// TIA Portal V20 export
FUNCTION_BLOCK "FB_FixtureUnloadLoad"   // FB65, SCL
{ S7_Optimized_Access := 'TRUE' }
// stored: MemoryReserve 100, SetENOAutomatically false
   VAR_INPUT
      iFixtureUnloadingRequest : Bool;
      iFixtureLoadingRequest : Bool;
      iFixtureBlowingRequest : Bool;
      iFixtureReleaseRequest : Bool;
      iFixtureV_InitRequest : Bool;
      iFixtureW_InitRequest : Bool;
      iWorkingModeFilling : Bool;
      iWorkingModeEmptying : Bool;
      iGripperReadyForUnloading : Bool;
      iGripperReadyForLoading : Bool;
      iGripperReadyForBlowing : Bool;
      iGripperReadyForRelease : Bool;
      iGripperReadyForV_Init : Bool;
      iGripperReadyForW_Init : Bool;
      iFixtureReadyForUnloading : Bool;
      iFixtureReadyForLoading : Bool;
      iFixtureReadyForBlowing : Bool;
      iFixtureReadyForRelease : Bool;
      iFixtureReadyForV_Init : Bool;
      iFixtureReadyForW_Init : Bool;
      iAxisReadyForUnloading : Bool;
      iAxisReadyForLoading : Bool;
      iAxisReadyForBlowing : Bool;
      iAxisReadyForRelease : Bool;
      iAxisReadyForV_Init : Bool;
      iAxisReadyForW_Init : Bool;
      iAxisV_W_Available : Bool;
   END_VAR
   VAR_OUTPUT
      oAxisV_W_Reservation : Bool;
      oNC_RID1 : Bool;
      oNC_RID2 : Bool;
   END_VAR
   VAR_IN_OUT
      ioFixtureUnloadingSeq : "UDT_SequenceInterface";
      ioFixtureLoadingSeq : "UDT_SequenceInterface";
      ioFixtureBlowingSeq : "UDT_SequenceInterface";
      ioFixtureReleaseSeq : "UDT_SequenceInterface";
      ioFixtureV_InitSeq : "UDT_SequenceInterface";
      ioFixtureW_InitSeq : "UDT_SequenceInterface";
   END_VAR
   VAR
      sRT_FixtureUnloadingRequest : R_TRIG;
      sRT_FixtureLoadingRequest { S7_SetPoint := 'True'} : R_TRIG;
      sRT_FixtureBlowingRequest { S7_SetPoint := 'True'} : R_TRIG;
      sRT_FixtureReleaseRequest { S7_SetPoint := 'True'} : R_TRIG;
      sRT_FixtureV_InitRequest { S7_SetPoint := 'True'} : R_TRIG;
      sRT_FixtureW_InitRequest { S7_SetPoint := 'True'} : R_TRIG;
      sMemoUnloadingRequest { S7_SetPoint := 'True'} : Bool;
      sMemoLoadingRequest { S7_SetPoint := 'True'} : Bool;
      sMemoBlowingRequest { S7_SetPoint := 'True'} : Bool;
      sMemoReleaseRequest { S7_SetPoint := 'True'} : Bool;
      sMemoV_InitRequest : Bool;
      sMemoW_InitRequest : Bool;
      sTONUnloadingNotFinished : TON_TIME;
      sTONBlowingNotFinished { S7_SetPoint := 'True'} : TON_TIME;
      sTONLoadingNotFinished { S7_SetPoint := 'True'} : TON_TIME;
   END_VAR
BEGIN
   REGION Description header 
       //==================================================================================
       // POSALUX Swiss SA / (C) Copyright 2026
       //----------------------------------------------------------------------------------
       // Title: FB_FixtureUnloadLoadMain
       // Comment/Function: 
       // Author: Fabien WALDT
       // Engineering: TIA Portal v20
       //----------------------------------------------------------------------------------
       // Change log table:
       // Version  | Date     | Expert in charge | Changes applied
       // ---------|----------|------------------|-----------------------------------------
       // 00.00.01 | 20260122 | WFA              | First released version
       // =================================================================================
   END_REGION

   REGION Init
       IF "LBP_Chan1".A_Reset THEN
           #oAxisV_W_Reservation := FALSE;
           #oNC_RID1 := FALSE;
           #oNC_RID2 := FALSE;
           #ioFixtureUnloadingSeq.StartRequest := FALSE;
           #ioFixtureLoadingSeq.StartRequest := FALSE;
           #ioFixtureBlowingSeq.StartRequest := FALSE;
           #ioFixtureReleaseSeq.StartRequest := FALSE;
           #ioFixtureV_InitSeq.StartRequest := FALSE;
           #ioFixtureW_InitSeq.StartRequest := FALSE;
           #sMemoUnloadingRequest := FALSE;
           #sMemoLoadingRequest := FALSE;
           #sMemoBlowingRequest := FALSE;
           #sMemoReleaseRequest := FALSE;
       END_IF;
   END_REGION

   REGION Fixture Unload Request
       #sRT_FixtureUnloadingRequest(CLK := #iFixtureUnloadingRequest        // M Code
                                    AND NOT #iWorkingModeFilling            // Not Mode Filling (No Part on Fixture)
                                    AND NOT (#iWorkingModeEmptying AND "DB_PartManagement".sPosition.sFixtureEmpty AND "DB_PartManagement".sPosition.sGripperEmpty)); // Not Gripper and Fixture Empty
       IF #sRT_FixtureUnloadingRequest.Q THEN
           #oNC_RID2 := TRUE;
           #sMemoUnloadingRequest := TRUE;
           "DB_LoaderFixtureMain".sBlowingNotFinished := FALSE;
           "DB_LoaderFixtureMain".sLoadingNotFinished := FALSE;
           "DB_LoaderFixtureMain".sUnloadingNotFinished := FALSE;
       END_IF;

       IF #sMemoUnloadingRequest
           AND #iGripperReadyForUnloading
           AND #iFixtureReadyForUnloading
           AND #iAxisReadyForUnloading
           AND NOT #iWorkingModeFilling
           AND NOT (#iWorkingModeEmptying AND "DB_PartManagement".sPosition.sFixtureEmpty AND "DB_PartManagement".sPosition.sGripperEmpty) THEN
           #oAxisV_W_Reservation := TRUE;
           #ioFixtureUnloadingSeq.StartRequest := TRUE;
       END_IF;

       #sTONUnloadingNotFinished(IN := "DB_LoaderFixtureMain".sUnloadingNotFinished,
                                 PT := T#100ms);

       IF #ioFixtureUnloadingSeq.JobDone
           OR "DB_LoaderFixtureMain".sUnloadingNotFinished THEN
           #ioFixtureUnloadingSeq.StartRequest := FALSE;
           #sMemoUnloadingRequest := FALSE;
       END_IF;

       IF #ioFixtureUnloadingSeq.JobDone
           OR #sTONUnloadingNotFinished.Q THEN
           #oNC_RID2 := FALSE;
       END_IF;
   END_REGION

   REGION Fixture Load Request
       #sRT_FixtureLoadingRequest(CLK := #iFixtureLoadingRequest
                                  AND NOT (#iWorkingModeEmptying AND NOT "DB_PartManagement".sPosition.sGripper.Undrilled.Presence.Part));
       IF #sRT_FixtureLoadingRequest.Q THEN
           #oNC_RID2 := TRUE;
           #sMemoLoadingRequest := TRUE;
           "DB_LoaderFixtureMain".sBlowingNotFinished := FALSE;
           "DB_LoaderFixtureMain".sLoadingNotFinished := FALSE;
           "DB_LoaderFixtureMain".sUnloadingNotFinished := FALSE;
       END_IF;

       IF #sMemoLoadingRequest
           AND #iGripperReadyForLoading
           AND #iFixtureReadyForLoading
           AND #iAxisReadyForLoading THEN
           #oAxisV_W_Reservation := TRUE;
           #ioFixtureLoadingSeq.StartRequest := TRUE;
       END_IF;

       #sTONLoadingNotFinished(IN := "DB_LoaderFixtureMain".sLoadingNotFinished,
                                 PT := T#100ms);

       IF #ioFixtureLoadingSeq.JobDone
           OR "DB_LoaderFixtureMain".sLoadingNotFinished THEN
           #ioFixtureLoadingSeq.StartRequest := FALSE;
           #sMemoLoadingRequest := FALSE;
       END_IF;

       IF #ioFixtureLoadingSeq.JobDone
           OR #sTONLoadingNotFinished.Q THEN
           #oNC_RID2 := FALSE;
       END_IF;
   END_REGION

   REGION Fixture Blowing Request
       #sRT_FixtureBlowingRequest(CLK := #iFixtureBlowingRequest
                                  AND NOT (#iWorkingModeEmptying AND NOT "DB_PartManagement".sPosition.sGripper.Undrilled.Presence.Part));
       IF #sRT_FixtureBlowingRequest.Q THEN
           #oNC_RID2 := TRUE;
           #sMemoBlowingRequest := TRUE;
           "DB_LoaderFixtureMain".sBlowingNotFinished := FALSE;
           "DB_LoaderFixtureMain".sLoadingNotFinished := FALSE;
           "DB_LoaderFixtureMain".sUnloadingNotFinished := FALSE;
       END_IF;

       IF #sMemoBlowingRequest
           AND #iGripperReadyForBlowing
           AND #iFixtureReadyForBlowing
           AND #iAxisReadyForBlowing THEN
           #oAxisV_W_Reservation := TRUE;
           #ioFixtureBlowingSeq.StartRequest := TRUE;
       END_IF;

       #sTONBlowingNotFinished(IN := "DB_LoaderFixtureMain".sBlowingNotFinished,
                               PT := T#100ms);

       IF #ioFixtureBlowingSeq.JobDone
       OR "DB_LoaderFixtureMain".sBlowingNotFinished THEN
           #ioFixtureBlowingSeq.StartRequest := FALSE;
           #sMemoBlowingRequest := FALSE;
       END_IF;

       IF #ioFixtureBlowingSeq.JobDone
           OR #sTONBlowingNotFinished.Q THEN
           #oNC_RID2 := FALSE;
       END_IF;
   END_REGION

   REGION Fixture Release Request
       #sRT_FixtureReleaseRequest(CLK := #iFixtureReleaseRequest
                                  OR #ioFixtureLoadingSeq.JobDone
                                  OR (#ioFixtureUnloadingSeq.JobDone AND (#iWorkingModeEmptying AND NOT "DB_PartManagement".sPosition.sGripper.Undrilled.Presence.Part)));
       // IF #sRT_FixtureReleaseRequest.Q THEN
       //     #oNC_RID2 := TRUE;
       //     #sMemoReleaseRequest := TRUE;
       // END_IF;

       IF (#sMemoReleaseRequest OR #ioFixtureLoadingSeq.JobDone
           OR (#ioFixtureUnloadingSeq.JobDone
           AND (#iWorkingModeEmptying AND NOT "DB_PartManagement".sPosition.sGripper.Undrilled.Presence.Part)))
           AND #iGripperReadyForRelease
           AND #iFixtureReadyForRelease
           AND #iAxisReadyForRelease THEN
           #oAxisV_W_Reservation := TRUE;
           #ioFixtureReleaseSeq.StartRequest := TRUE;
       END_IF;

       IF #ioFixtureReleaseSeq.JobDone
       OR "DB_LoaderFixtureMain".sReleaseNotFinished THEN
           #ioFixtureReleaseSeq.StartRequest := FALSE;
           #sMemoReleaseRequest := FALSE;
           #oNC_RID2 := FALSE;
           #oAxisV_W_Reservation := FALSE;
       END_IF;
   END_REGION

   REGION V Init Request
       #sRT_FixtureV_InitRequest(CLK := #iFixtureV_InitRequest);
       IF #sRT_FixtureV_InitRequest.Q THEN
           #oNC_RID1 := TRUE;
           #sMemoV_InitRequest := TRUE;
       END_IF;

       IF #sMemoV_InitRequest
           AND #iGripperReadyForV_Init
           AND #iFixtureReadyForV_Init
           AND #iAxisReadyForV_Init THEN
               #oAxisV_W_Reservation := TRUE;
               #ioFixtureV_InitSeq.StartRequest := TRUE;
       END_IF;

       IF #ioFixtureV_InitSeq.JobDone
       OR "DB_LoaderFixtureMain".sV_InitNotFinished THEN
           #ioFixtureV_InitSeq.StartRequest := FALSE;
           #sMemoV_InitRequest := FALSE;
           #oNC_RID1 := FALSE;
           #oAxisV_W_Reservation := FALSE;
       END_IF;
   END_REGION

   REGION W Init Request
       #sRT_FixtureW_InitRequest(CLK := #iFixtureW_InitRequest);
       IF #sRT_FixtureW_InitRequest.Q THEN
           #oNC_RID1 := TRUE;
           #sMemoW_InitRequest := TRUE;
       END_IF;

       IF #sMemoW_InitRequest
           AND #iGripperReadyForW_Init
           AND #iFixtureReadyForW_Init
           AND #iAxisReadyForW_Init THEN
           #oAxisV_W_Reservation := TRUE;
           #ioFixtureW_InitSeq.StartRequest := TRUE;
       END_IF;

       IF #ioFixtureW_InitSeq.JobDone
       OR "DB_LoaderFixtureMain".sW_InitNotFinished THEN
           #ioFixtureW_InitSeq.StartRequest := FALSE;
           #sMemoW_InitRequest := FALSE;
           #oNC_RID1 := FALSE;
           #oAxisV_W_Reservation := FALSE;
       END_IF;
   END_REGION
END_FUNCTION_BLOCK
